{attribute 'OPC.UA.DA.StructuredType' := '1'}
TYPE ST_JanitzaState :
STRUCT
	fPower 					: REAL;
	sPowerUnit				: STRING := 'kW';
END_STRUCT
END_TYPE

(* stored: Version 1.1.0.1, ProductVersion 3.1.4024.10
   DUT ST_JanitzaState: Id {e606aa29-d82c-4475-a253-4d230cc24865} *)
